// Mitsubishi GX Works2 project: On_thi_Tot_Nghiep   PLC: FX2N/FX2NC

PROGRAM MAIN
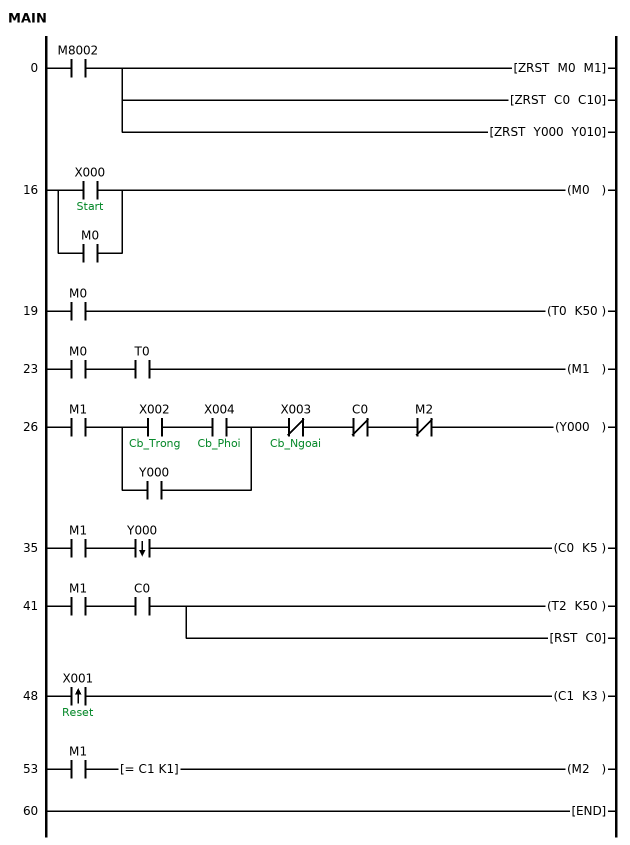
0     LD      M8002
      ZRST    M0 M1
      ZRST    C0 C10
      ZRST    Y000 Y010
16    LD      X000  ; Start
      OR      M0
      OUT     M0
19    LD      M0
      OUT     T0 K50
23    LD      M0
      AND     T0
      OUT     M1
26    LD      M1
      LD      X002  ; Cb_Trong
      AND     X004  ; Cb_Phoi
      OR      Y000
      ANB
      ANI     X003  ; Cb_Ngoai
      ANI     C0
      ANI     M2
      OUT     Y000
35    LD      M1
      ANDF    Y000
      OUT     C0 K5
41    LD      M1
      AND     C0
      OUT     T2 K50
      RST     C0
48    LDP     X001  ; Reset
      OUT     C1 K3
53    LD      M1
      AND=    C1 K1
      OUT     M2
60    END
END_PROGRAM
